FUNCTION_BLOCK ABSTRACT AngleSequenceAccessor EXTENDS Matrix
VAR_INPUT
END_VAR
VAR_OUTPUT
END_VAR
VAR
	O_ : REFERENCE TO AngleSequenceOrientation;
END_VAR

//Total number of columns in this matrix
PROPERTY PUBLIC Cols : UINT
GET
IF NOT __ISVALIDREF(O_) THEN
	Cols := 0;
	LogWarning('%s Attempted Cols access using uninitialized Matrix Accessor');
ELSE
	Cols :=1;
END_IF
END_GET
END_PROPERTY

METHOD PUBLIC Init
VAR_INPUT
	O : REFERENCE TO AngleSequenceOrientation;
END_VAR
O_ REF= O;
END_METHOD

//Total number of rows in this matrix
PROPERTY PUBLIC Rows : UINT
GET
IF NOT __ISVALIDREF(O_) THEN
	Rows := 0;
	LogWarning('%s Attempted Rows access using uninitialized Matrix Accessor');
ELSE
	Rows := O_.Length;
END_IF;
END_GET
END_PROPERTY

END_FUNCTION_BLOCK

(* stored: Version 1.1.0.1, ProductVersion 3.1.4024.9
   POU AngleSequenceAccessor: Id {55367483-4f8f-07ac-3649-8652ccddc0d4}, SpecialFunc None
   Folder Initialziers: Id {79a0317c-0b4a-09d0-2d30-fb28beb622f5}
   Folder Overrides: Id {08eb1a25-3c5b-0a78-0cf3-93f51fb93b13}
   Property Cols: Id {36d083b3-08b3-0294-1c57-7ba1fc67cb70}
   Get Get: Id {db991d45-12c9-071b-3e38-f092cfeb5cb6}
   Method Init: Id {23575e2e-d16b-0e28-2710-d6c820171276}
   Property Rows: Id {3dc241e7-7a77-02e2-2af7-2f2db64f9fe1}
   Get Get: Id {5d12b961-486d-019d-287d-991e68701dd3} *)
